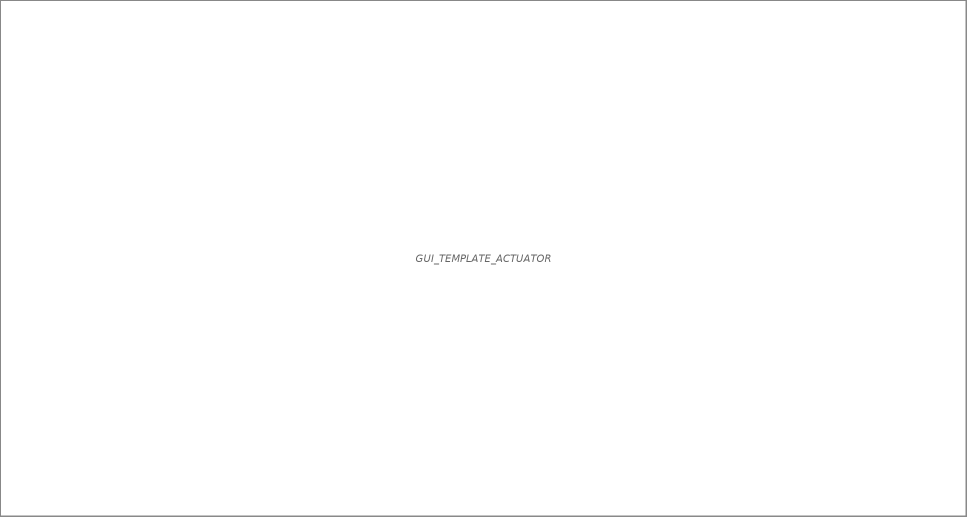
VISUALIZATION GUI_Actuator002  // 967x517
    Frame (0,0 967x517)
        shows GUI_TEMPLATE_ACTUATOR(m_Instance := MAIN.Actuator002)
END_VISUALIZATION

(* stored: Version 1.1.0.1, ProductVersion 3.1.4024.3
   Visu GUI_Actuator002: Id {6564160e-88ed-4e89-ac3e-ea6d0393238f} *)
